// TIA Portal V20 export
FUNCTION_BLOCK "Side_Driver"   // FB2, LAD
{ S7_Optimized_Access := 'TRUE' }
// stored: MemoryReserve 100, SetENOAutomatically false
   VAR_INPUT
      Reset : Bool;
      Jog_Forward_SL : Bool;
      Jog_Forward_SR : Bool;
      Jog_Backward_SL : Bool;
      Jog_Backward_SR : Bool;
      Set_SL_Speed : Int;
      Set_SR_Speed : Int;
      Set_Acc : Int;
      Set_Dcc : Int;
      HWIdentSL : HW_IO;
      HWIdentSR : HW_IO;
   END_VAR
   VAR_OUTPUT
      oSL_Communication_OK : Bool;
      oSR_Communication_OK : Bool;
      oSL_Forward_Flag : Bool;
      oSL_Backward_Flag : Bool;
      oSR_Forward_Flag : Bool;
      oSR_Backward_Flag : Bool;
      oError : Bool;
   END_VAR
   VAR_IN_OUT
      iSL_Drive_Param : "SEW_MOVIKIT_VelocityDrive_SETPOINTS_V2.1";
      iSR_Drive_Param : "SEW_MOVIKIT_VelocityDrive_SETPOINTS_V2.1";
      oSL_Drive_Param : "SEW_MOVIKIT_VelocityDrive_STATUS_V2.1";
      oSR_Drive_Param : "SEW_MOVIKIT_VelocityDrive_STATUS_V2.1";
   END_VAR
   VAR
      Error_SL : Bool;
      Error_SR : Bool;
   END_VAR
   VAR_TEMP
      Speed_SL_reverse : Int;
      Speed_SR_reverse : Int;
   END_VAR
   VAR_TEMP   // added for the SCL form of the ladder/FBD networks
      _w1 : Bool;
   END_VAR
BEGIN

REGION Network 1: SL Movikit
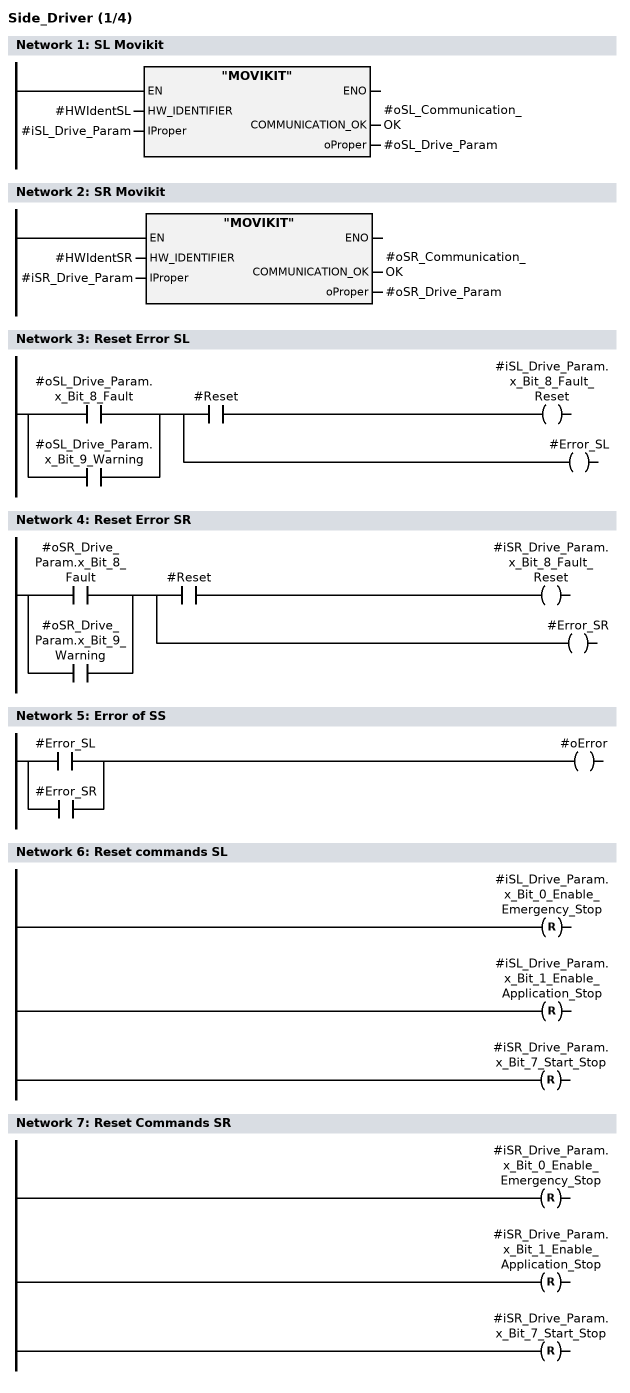
   RUNG wire#powerrail
      "MOVIKIT"(HW_IDENTIFIER := #HWIdentSL, IProper := #iSL_Drive_Param, COMMUNICATION_OK => #oSL_Communication_OK, oProper => #oSL_Drive_Param)
   END_RUNG
   // the same network as SCL:
   "MOVIKIT"(HW_IDENTIFIER := #HWIdentSL,
             IProper := #iSL_Drive_Param,
             COMMUNICATION_OK => #oSL_Communication_OK,
             oProper => #oSL_Drive_Param);
END_REGION

REGION Network 2: SR Movikit
   RUNG wire#powerrail
      "MOVIKIT"(HW_IDENTIFIER := #HWIdentSR, IProper := #iSR_Drive_Param, COMMUNICATION_OK => #oSR_Communication_OK, oProper => #oSR_Drive_Param)
   END_RUNG
   // the same network as SCL:
   "MOVIKIT"(HW_IDENTIFIER := #HWIdentSR,
             IProper := #iSR_Drive_Param,
             COMMUNICATION_OK => #oSR_Communication_OK,
             oProper => #oSR_Drive_Param);
END_REGION

REGION Network 3: Reset Error SL
   RUNG wire#powerrail
      Contact( #oSL_Drive_Param.x_Bit_8_Fault )
      wire#w1
      Contact( #Reset )
      Coil( #iSL_Drive_Param.x_Bit_8_Fault_Reset )
   END_RUNG
   RUNG wire#powerrail
      Contact( #oSL_Drive_Param.x_Bit_9_Warning )
   END_RUNG wire#w1
   RUNG wire#w1
      Coil( #Error_SL )
   END_RUNG
   // the same network as SCL:
   #_w1 := #oSL_Drive_Param.x_Bit_8_Fault OR #oSL_Drive_Param.x_Bit_9_Warning;
   #iSL_Drive_Param.x_Bit_8_Fault_Reset := #_w1 AND #Reset;
   #Error_SL := #_w1;
END_REGION

REGION Network 4: Reset Error SR
   RUNG wire#powerrail
      Contact( #oSR_Drive_Param.x_Bit_8_Fault )
      wire#w1
      Contact( #Reset )
      Coil( #iSR_Drive_Param.x_Bit_8_Fault_Reset )
   END_RUNG
   RUNG wire#powerrail
      Contact( #oSR_Drive_Param.x_Bit_9_Warning )
   END_RUNG wire#w1
   RUNG wire#w1
      Coil( #Error_SR )
   END_RUNG
   // the same network as SCL:
   #_w1 := #oSR_Drive_Param.x_Bit_8_Fault OR #oSR_Drive_Param.x_Bit_9_Warning;
   #iSR_Drive_Param.x_Bit_8_Fault_Reset := #_w1 AND #Reset;
   #Error_SR := #_w1;
END_REGION

REGION Network 5: Error of SS
   RUNG wire#powerrail
      Contact( #Error_SL )
      wire#w1
      Coil( #oError )
   END_RUNG
   RUNG wire#powerrail
      Contact( #Error_SR )
   END_RUNG wire#w1
   // the same network as SCL:
   #oError := #Error_SL OR #Error_SR;
END_REGION

REGION Network 6: Reset commands SL
   RUNG wire#powerrail
      R_Coil( #iSL_Drive_Param.x_Bit_0_Enable_Emergency_Stop )
   END_RUNG
   RUNG wire#powerrail
      R_Coil( #iSL_Drive_Param.x_Bit_1_Enable_Application_Stop )
   END_RUNG
   RUNG wire#powerrail
      R_Coil( #iSR_Drive_Param.x_Bit_7_Start_Stop )
   END_RUNG
   // the same network as SCL:
   #iSL_Drive_Param.x_Bit_0_Enable_Emergency_Stop := FALSE;
   #iSL_Drive_Param.x_Bit_1_Enable_Application_Stop := FALSE;
   #iSR_Drive_Param.x_Bit_7_Start_Stop := FALSE;
END_REGION

REGION Network 7: Reset Commands SR
   RUNG wire#powerrail
      R_Coil( #iSR_Drive_Param.x_Bit_0_Enable_Emergency_Stop )
   END_RUNG
   RUNG wire#powerrail
      R_Coil( #iSR_Drive_Param.x_Bit_1_Enable_Application_Stop )
   END_RUNG
   RUNG wire#powerrail
      R_Coil( #iSR_Drive_Param.x_Bit_7_Start_Stop )
   END_RUNG
   // the same network as SCL:
   #iSR_Drive_Param.x_Bit_0_Enable_Emergency_Stop := FALSE;
   #iSR_Drive_Param.x_Bit_1_Enable_Application_Stop := FALSE;
   #iSR_Drive_Param.x_Bit_7_Start_Stop := FALSE;
END_REGION

REGION Network 8: Reverse directions
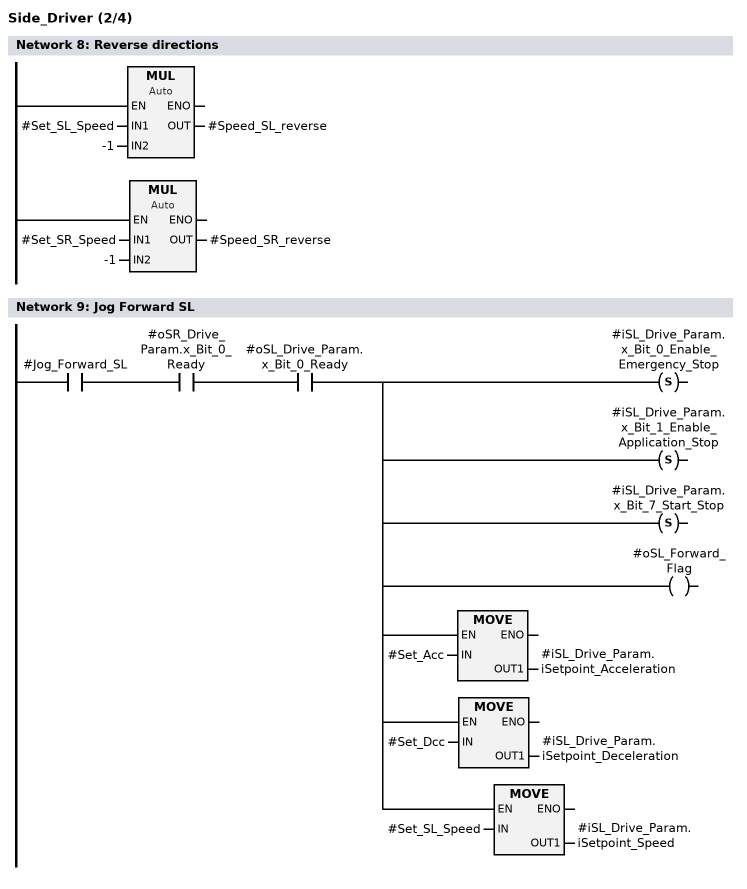
   RUNG wire#powerrail
      Mul(in1 := #Set_SL_Speed, in2 := -1, out => #Speed_SL_reverse)
   END_RUNG
   RUNG wire#powerrail
      Mul(in1 := #Set_SR_Speed, in2 := -1, out => #Speed_SR_reverse)
   END_RUNG
   // the same network as SCL:
   #Speed_SL_reverse := #Set_SL_Speed * (-1);
   #Speed_SR_reverse := #Set_SR_Speed * (-1);
END_REGION

REGION Network 9: Jog Forward SL
   RUNG wire#powerrail
      Contact( #Jog_Forward_SL )
      Contact( #oSR_Drive_Param.x_Bit_0_Ready )
      Contact( #oSL_Drive_Param.x_Bit_0_Ready )
      wire#w1
      S_Coil( #iSL_Drive_Param.x_Bit_0_Enable_Emergency_Stop )
   END_RUNG
   RUNG wire#w1
      S_Coil( #iSL_Drive_Param.x_Bit_1_Enable_Application_Stop )
   END_RUNG
   RUNG wire#w1
      S_Coil( #iSL_Drive_Param.x_Bit_7_Start_Stop )
   END_RUNG
   RUNG wire#w1
      Coil( #oSL_Forward_Flag )
   END_RUNG
   RUNG wire#w1
      Move(in := #Set_Acc, out1 => #iSL_Drive_Param.iSetpoint_Acceleration)
   END_RUNG
   RUNG wire#w1
      Move(in := #Set_Dcc, out1 => #iSL_Drive_Param.iSetpoint_Deceleration)
   END_RUNG
   RUNG wire#w1
      Move(in := #Set_SL_Speed, out1 => #iSL_Drive_Param.iSetpoint_Speed)
   END_RUNG
   // the same network as SCL:
   #_w1 := #Jog_Forward_SL AND #oSR_Drive_Param.x_Bit_0_Ready AND #oSL_Drive_Param.x_Bit_0_Ready;
   IF #_w1 THEN
       #iSL_Drive_Param.x_Bit_0_Enable_Emergency_Stop := TRUE;
       #iSL_Drive_Param.x_Bit_1_Enable_Application_Stop := TRUE;
       #iSL_Drive_Param.x_Bit_7_Start_Stop := TRUE;
   END_IF;
   #oSL_Forward_Flag := #_w1;
   IF #_w1 THEN
       #iSL_Drive_Param.iSetpoint_Acceleration := #Set_Acc;
       #iSL_Drive_Param.iSetpoint_Deceleration := #Set_Dcc;
       #iSL_Drive_Param.iSetpoint_Speed := #Set_SL_Speed;
   END_IF;
END_REGION

REGION Network 10: Jog backward SL
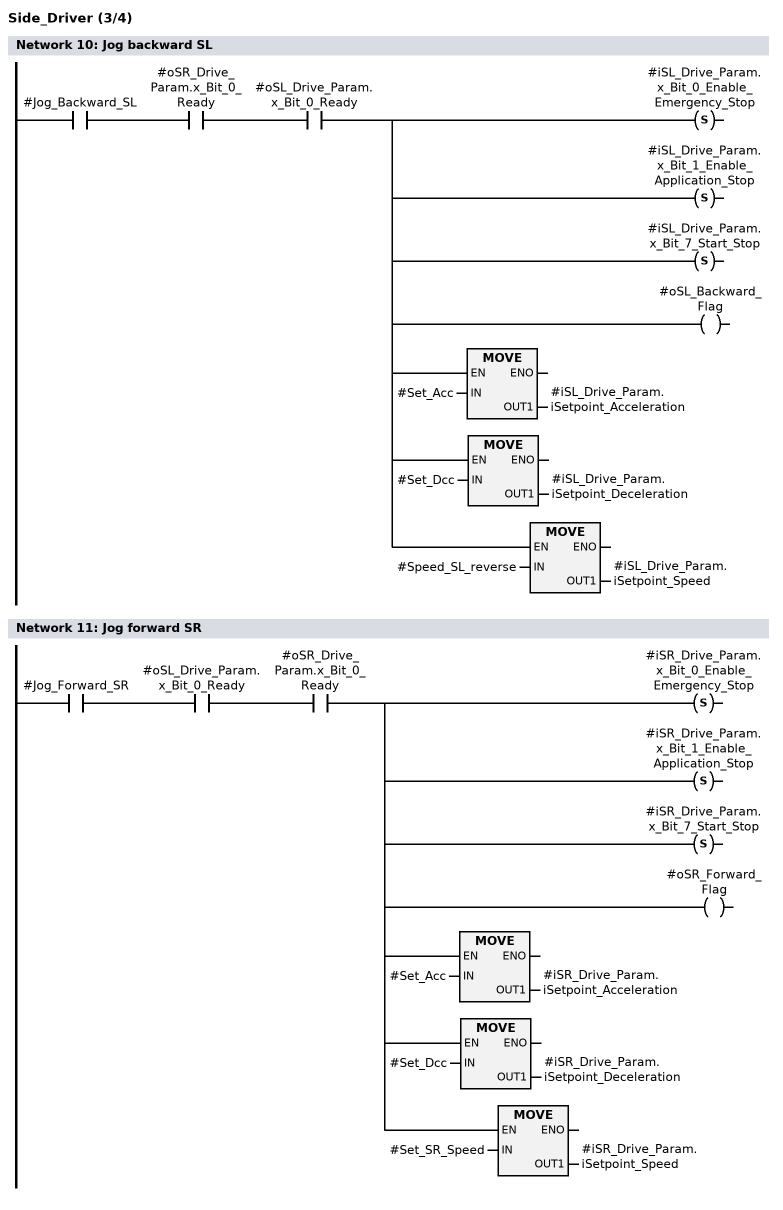
   RUNG wire#powerrail
      Contact( #Jog_Backward_SL )
      Contact( #oSR_Drive_Param.x_Bit_0_Ready )
      Contact( #oSL_Drive_Param.x_Bit_0_Ready )
      wire#w1
      S_Coil( #iSL_Drive_Param.x_Bit_0_Enable_Emergency_Stop )
   END_RUNG
   RUNG wire#w1
      S_Coil( #iSL_Drive_Param.x_Bit_1_Enable_Application_Stop )
   END_RUNG
   RUNG wire#w1
      S_Coil( #iSL_Drive_Param.x_Bit_7_Start_Stop )
   END_RUNG
   RUNG wire#w1
      Coil( #oSL_Backward_Flag )
   END_RUNG
   RUNG wire#w1
      Move(in := #Set_Acc, out1 => #iSL_Drive_Param.iSetpoint_Acceleration)
   END_RUNG
   RUNG wire#w1
      Move(in := #Set_Dcc, out1 => #iSL_Drive_Param.iSetpoint_Deceleration)
   END_RUNG
   RUNG wire#w1
      Move(in := #Speed_SL_reverse, out1 => #iSL_Drive_Param.iSetpoint_Speed)
   END_RUNG
   // the same network as SCL:
   #_w1 := #Jog_Backward_SL AND #oSR_Drive_Param.x_Bit_0_Ready AND #oSL_Drive_Param.x_Bit_0_Ready;
   IF #_w1 THEN
       #iSL_Drive_Param.x_Bit_0_Enable_Emergency_Stop := TRUE;
       #iSL_Drive_Param.x_Bit_1_Enable_Application_Stop := TRUE;
       #iSL_Drive_Param.x_Bit_7_Start_Stop := TRUE;
   END_IF;
   #oSL_Backward_Flag := #_w1;
   IF #_w1 THEN
       #iSL_Drive_Param.iSetpoint_Acceleration := #Set_Acc;
       #iSL_Drive_Param.iSetpoint_Deceleration := #Set_Dcc;
       #iSL_Drive_Param.iSetpoint_Speed := #Speed_SL_reverse;
   END_IF;
END_REGION

REGION Network 11: Jog forward SR
   RUNG wire#powerrail
      Contact( #Jog_Forward_SR )
      Contact( #oSL_Drive_Param.x_Bit_0_Ready )
      Contact( #oSR_Drive_Param.x_Bit_0_Ready )
      wire#w1
      S_Coil( #iSR_Drive_Param.x_Bit_0_Enable_Emergency_Stop )
   END_RUNG
   RUNG wire#w1
      S_Coil( #iSR_Drive_Param.x_Bit_1_Enable_Application_Stop )
   END_RUNG
   RUNG wire#w1
      S_Coil( #iSR_Drive_Param.x_Bit_7_Start_Stop )
   END_RUNG
   RUNG wire#w1
      Coil( #oSR_Forward_Flag )
   END_RUNG
   RUNG wire#w1
      Move(in := #Set_Acc, out1 => #iSR_Drive_Param.iSetpoint_Acceleration)
   END_RUNG
   RUNG wire#w1
      Move(in := #Set_Dcc, out1 => #iSR_Drive_Param.iSetpoint_Deceleration)
   END_RUNG
   RUNG wire#w1
      Move(in := #Set_SR_Speed, out1 => #iSR_Drive_Param.iSetpoint_Speed)
   END_RUNG
   // the same network as SCL:
   #_w1 := #Jog_Forward_SR AND #oSL_Drive_Param.x_Bit_0_Ready AND #oSR_Drive_Param.x_Bit_0_Ready;
   IF #_w1 THEN
       #iSR_Drive_Param.x_Bit_0_Enable_Emergency_Stop := TRUE;
       #iSR_Drive_Param.x_Bit_1_Enable_Application_Stop := TRUE;
       #iSR_Drive_Param.x_Bit_7_Start_Stop := TRUE;
   END_IF;
   #oSR_Forward_Flag := #_w1;
   IF #_w1 THEN
       #iSR_Drive_Param.iSetpoint_Acceleration := #Set_Acc;
       #iSR_Drive_Param.iSetpoint_Deceleration := #Set_Dcc;
       #iSR_Drive_Param.iSetpoint_Speed := #Set_SR_Speed;
   END_IF;
END_REGION

REGION Network 12: Jog Backward SR
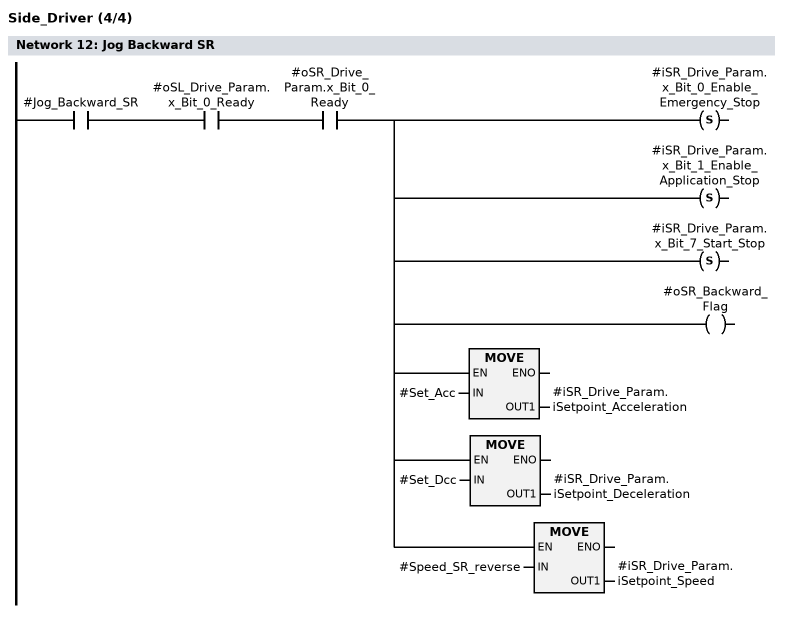
   RUNG wire#powerrail
      Contact( #Jog_Backward_SR )
      Contact( #oSL_Drive_Param.x_Bit_0_Ready )
      Contact( #oSR_Drive_Param.x_Bit_0_Ready )
      wire#w1
      S_Coil( #iSR_Drive_Param.x_Bit_0_Enable_Emergency_Stop )
   END_RUNG
   RUNG wire#w1
      S_Coil( #iSR_Drive_Param.x_Bit_1_Enable_Application_Stop )
   END_RUNG
   RUNG wire#w1
      S_Coil( #iSR_Drive_Param.x_Bit_7_Start_Stop )
   END_RUNG
   RUNG wire#w1
      Coil( #oSR_Backward_Flag )
   END_RUNG
   RUNG wire#w1
      Move(in := #Set_Acc, out1 => #iSR_Drive_Param.iSetpoint_Acceleration)
   END_RUNG
   RUNG wire#w1
      Move(in := #Set_Dcc, out1 => #iSR_Drive_Param.iSetpoint_Deceleration)
   END_RUNG
   RUNG wire#w1
      Move(in := #Speed_SR_reverse, out1 => #iSR_Drive_Param.iSetpoint_Speed)
   END_RUNG
   // the same network as SCL:
   #_w1 := #Jog_Backward_SR AND #oSL_Drive_Param.x_Bit_0_Ready AND #oSR_Drive_Param.x_Bit_0_Ready;
   IF #_w1 THEN
       #iSR_Drive_Param.x_Bit_0_Enable_Emergency_Stop := TRUE;
       #iSR_Drive_Param.x_Bit_1_Enable_Application_Stop := TRUE;
       #iSR_Drive_Param.x_Bit_7_Start_Stop := TRUE;
   END_IF;
   #oSR_Backward_Flag := #_w1;
   IF #_w1 THEN
       #iSR_Drive_Param.iSetpoint_Acceleration := #Set_Acc;
       #iSR_Drive_Param.iSetpoint_Deceleration := #Set_Dcc;
       #iSR_Drive_Param.iSetpoint_Speed := #Speed_SR_reverse;
   END_IF;
END_REGION
END_FUNCTION_BLOCK
